{attribute 'conditionalshow'}
FUNCTION_BLOCK FB_CV_DINT_TO_WORD
VAR_INPUT
	{attribute 'hide'}
	diInputValue				: DINT;								//Input value that is converted into the output value
	{attribute 'hide'}
	eByteOrderForConvert		: eByteOrder;						//Byte Format							
END_VAR
VAR_OUTPUT
	{attribute 'hide'}
	wOutputValue_1				: WORD;								//Converted output value
	{attribute 'hide'}
	wOutputValue_2				: WORD;								//Converted output value
END_VAR
VAR
END_VAR

//Creator : Kai Ebensperger
//Company : Lynus AG
//Date : 28.04.2021
//Version : 1.0.0.0

//With this functionblock its possible to convert a certain Datatyp in a other Datatype
//The byte order can be selected between BigEndian and LittleEndian
//DINT TO WORD
//Created for the Edge Device Lib over Modbus TCP
//Modbus TCP is WORD oriented

IF eByteOrderForConvert = eByteOrder.eBigEndian THEN
	wOutputValue_1 := DWORD_TO_WORD(SHR(DINT_TO_DWORD(diInputValue),16) AND 16#FFFF);
	wOutputValue_2 := DWORD_TO_WORD(DINT_TO_DWORD(diInputValue)) AND 16#FFFF;
ELSE
	wOutputValue_2 := DWORD_TO_WORD(SHR(DINT_TO_DWORD(diInputValue),16) AND 16#FFFF);
	wOutputValue_1 := DWORD_TO_WORD(DINT_TO_DWORD(diInputValue)) AND 16#FFFF;
END_IF

END_FUNCTION_BLOCK

(* stored: Version 1.1.0.1, ProductVersion 3.1.4024.9
   POU FB_CV_DINT_TO_WORD: Id {8f3cd839-b7b0-4be3-ac26-e7041a480581}, SpecialFunc None *)
